// Mitsubishi GX Works2 project: z05   PLC: Q02/Q02H

PROGRAM MAIN
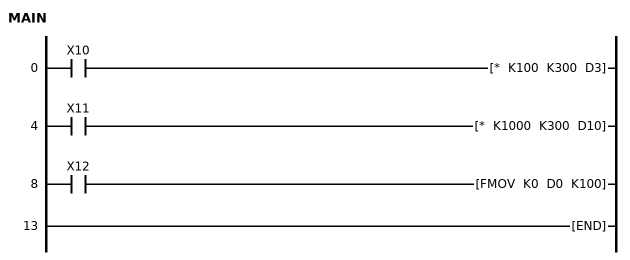
0     LD      X10
      *       K100 K300 D3
4     LD      X11
      *       K1000 K300 D10
8     LD      X12
      FMOV    K0 D0 K100
13    END
END_PROGRAM
